{attribute 'linkalways'} 
{attribute 'no_explicit_call' := 'This FB is a CLASS and must be accessed using methods or properties'}
{attribute 'enable_dynamic_creation'}
FUNCTION_BLOCK _ETcVnWorldCoordinateSystem EXTENDS EnumDatatypeBase
VAR
	localData : ETcVnWorldCoordinateSystem;
	activeData : REFERENCE TO ETcVnWorldCoordinateSystem;
	enumBaseDatatype : _DINT(localData);
END_VAR

METHOD PRIVATE AddLocalEnumeration
VAR_INPUT
	Enumeration : T_MAXSTRING;
	Value : ETcVnWorldCoordinateSystem;
END_VAR
AddEnumeration(Enumeration, Value);
END_METHOD

PROPERTY PUBLIC Address : PVOID
GET
Address := ADR(activeData);
END_GET
END_PROPERTY

METHOD PUBLIC ClearReference
VAR_INPUT
END_VAR
activeData REF= localData;
SetBaseDatatypeReference();
END_METHOD

METHOD PUBLIC Clone : I_Datatype
VAR
    pClone : POINTER TO _ETcVnWorldCoordinateSystem;
END_VAR
pClone := __NEW(_ETcVnWorldCoordinateSystem(InitialValue := Value));
Clone := pClone^;
END_METHOD

METHOD FB_init : BOOL
VAR_INPUT
	bInitRetains : BOOL; // if TRUE, the retain variables are initialized (warm start / cold start)
	bInCopyCode : BOOL;  // if TRUE, the instance afterwards gets moved into the copy code (online change)
	InitialValue : ETcVnWorldCoordinateSystem;
END_VAR
localData := InitialValue;
AddBaseDatatype(enumBaseDatatype);
ClearReference();

AddLocalEnumeration('TCVN_WCS_X_RIGHT_Y_DOWN' , ETcVnWorldCoordinateSystem.TCVN_WCS_X_RIGHT_Y_DOWN);
AddLocalEnumeration('TCVN_WCS_X_DOWN_Y_RIGHT', ETcVnWorldCoordinateSystem.TCVN_WCS_X_DOWN_Y_RIGHT);
AddLocalEnumeration('TCVN_WCS_X_LEFT_Y_DOWN', ETcVnWorldCoordinateSystem.TCVN_WCS_X_LEFT_Y_DOWN);
AddLocalEnumeration('TCVN_WCS_X_UP_Y_RIGHT', ETcVnWorldCoordinateSystem.TCVN_WCS_X_UP_Y_RIGHT);
AddLocalEnumeration('TCVN_WCS_X_RIGHT_Y_UP', ETcVnWorldCoordinateSystem.TCVN_WCS_X_RIGHT_Y_UP);
AddLocalEnumeration('TCVN_WCS_X_DOWN_Y_LEFT', ETcVnWorldCoordinateSystem.TCVN_WCS_X_DOWN_Y_LEFT);
AddLocalEnumeration('TCVN_WCS_X_LEFT_Y_UP', ETcVnWorldCoordinateSystem.TCVN_WCS_X_LEFT_Y_UP);
AddLocalEnumeration('TCVN_WCS_X_UP_Y_LEFT', ETcVnWorldCoordinateSystem.TCVN_WCS_X_UP_Y_LEFT);
END_METHOD

PROPERTY PUBLIC Identifier : T_MAXSTRING
GET
Identifier := 'ETcVnWorldCoordinateSystem';
END_GET
END_PROPERTY

METHOD IsEnumeratorValueEqual : BOOL
VAR_INPUT
	Enumerator : I_KeyValueForwardEnumerator;
END_VAR
VAR
	storedValue : ETcVnWorldCoordinateSystem;
END_VAR
IF NOT Enumerator.TryGet(storedValue) THEN
	RETURN;
END_IF

IsEnumeratorValueEqual := storedValue = activeData;
END_METHOD

METHOD PUBLIC MakeReferenceTo
VAR_INPUT
	ReferenceTarget : REFERENCE TO ETcVnWorldCoordinateSystem;
END_VAR
activeData REF= ReferenceTarget;
SetBaseDatatypeReference();
END_METHOD

METHOD PROTECTED SetBaseDatatypeReference
VAR_INPUT
END_VAR
enumBaseDatatype.MakeReferenceTo(activeData);
END_METHOD

PROPERTY PUBLIC Size : UDINT
GET
Size := SIZEOF(activeData);
END_GET
END_PROPERTY

METHOD TryMakeReferenceTo : BOOL
VAR_INPUT
	Target : I_Datatype;
END_VAR
VAR
	targetAsEnum : I_EnumDatatype;
	pTargetData : POINTER TO ETcVnWorldCoordinateSystem;
END_VAR
IF NOT Target.TryResolveAsEnumDatatype(targetAsEnum) THEN
	RETURN;
END_IF

IF targetAsEnum.Identifier <> Identifier THEN
	RETURN;
END_IF

pTargetData := Target.Address;
activeData REF= pTargetData^;
SetBaseDatatypeReference();
TryMakeReferenceTo := TRUE;
END_METHOD

PROPERTY PUBLIC Value : ETcVnWorldCoordinateSystem
GET
Value := activeData;
END_GET
SET
activeData := Value;
END_SET
END_PROPERTY

END_FUNCTION_BLOCK

(* stored: Version 1.1.0.1
   POU _ETcVnWorldCoordinateSystem: Id {985d5a3c-3841-4c89-a706-748a3e4d6e77}, SpecialFunc None
   Folder Constructor: Id {00922633-5122-4b52-a7be-121bdae41642}
   Folder Private: Id {1a3b1399-b548-4b7f-beef-7981c77cf7be}
   Folder Protected: Id {9b5b3916-d4a9-4475-8b61-5e1d1906a351}
   Method AddLocalEnumeration: Id {e785990b-55ba-4b30-b79e-700a882c4088}
   Property Address: Id {21fe4155-76bb-4565-9955-a1bfe7fbcc08}
   Get Get: Id {ba9786d0-65ff-471a-91f9-00d928cd5807}
   Method ClearReference: Id {2dbcaf50-3897-4f87-b19c-a4758ec20c89}
   Method Clone: Id {cd7fcfd3-5577-4688-aea3-a1bed688fa14}
   Method FB_init: Id {b9000f8c-7cdc-461c-9661-b5da7ec8b4dd}
   Property Identifier: Id {6e006b05-8c39-404a-97ae-9789f5b41cea}
   Get Get: Id {2702133b-63d8-496e-8a51-782626224725}
   Method IsEnumeratorValueEqual: Id {3592fded-abdd-4fee-b2af-1497f77ce44f}
   Method MakeReferenceTo: Id {af54acee-aba6-4811-9276-110c9b7b9c60}
   Method SetBaseDatatypeReference: Id {3f2c82cb-7b89-4ec9-b1e6-e46b79932765}
   Property Size: Id {0172ab05-8d77-46cd-8df5-fbc92d94b060}
   Get Get: Id {d958f5aa-a2e4-44e0-aa9a-1144d13a2d27}
   Method TryMakeReferenceTo: Id {7c569d35-dcfa-4d8d-900f-eb6cc7718567}
   Property Value: Id {da636c4e-dd4e-4a12-9d08-0981d9b0d3b1}
   Get Get: Id {a7671c34-6602-4bbe-bdcc-8b0aee52806c}
   Set Set: Id {e8a20f6c-4598-424b-8067-ec2e009c9677} *)
